// TIA Portal V20 export
DATA_BLOCK "IDB_Segments_Status"   // DB45
// stored: InstanceOfName ProductionLine.FB_Segments, InstanceOfType FB, Namespace ProductionLine
"ProductionLine.FB_Segments"
   // VAR
   //    ConveyorID : Int;
   //    "Counter" : Int;
   //    FlowRackLoop1 : Array[_."B1.1.1".._."B1.23.1"] of Bool;
   //    FlowRackLoop2 : Array[_."B1.6.1".._."B1.18.1"] of Bool;
   //    Fragileloop1 : Array[_."D1.1.1".._."E1.6.1"] of Bool;
   //    Fragileloop2 : Array[_."D1.9.1".._."D1.10.1"] of Bool;
   //    cmp : Struct
   //       FlowRackLoop1 : Array[_."B1.1.1".._."B1.23.1"] of Bool;
   //       FlowRackLoop2 : Array[_."B1.6.1".._."B1.18.1"] of Bool;
   //       Fragileloop1 : Array[_."D1.1.1".._."E1.6.1"] of Bool;
   //       Fragileloop2 : Array[_."D1.9.1".._."D1.10.1"] of Bool;
   //    END_STRUCT;
   //    FlowRackLoopReadyToRun : Bool;
   //    FlowRackWorkPlaceLeftReadyToRun : Bool;
   //    FlowRackWorkPlaceRightReadyToRun : Bool;
   //    FragileloopReadyToRun : Bool;
   // END_VAR
BEGIN
END_DATA_BLOCK
